(* IEC 61131-3 sources: ics/BLR101_ProenixContact/BLR101_5_ILC171_44/LogicalPOUs/MTR, 3 files *)

(* ---- MotorFB.ST ---- *)
(*@PROPERTIES_EX@
TYPE: POU
LOCALE: 0
IEC_LANGUAGE: ST
PLC_TYPE: independent
PROC_TYPE: independent
GROUP: MTRS.FB
*)
(*@KEY@:DESCRIPTION*)

(*@KEY@:END_DESCRIPTION*)
FUNCTION_BLOCK MotorFB

(*Group:Default*)

VAR_IN_OUT
	Mot_strct :	MTR;
	Aux_strct :	MTR_MISC;
END_VAR

VAR_INPUT
	Cycle :	CCL;
END_VAR

VAR_EXTERNAL
	TICK_1S_PLS :	BOOL;
END_VAR

VAR_OUTPUT
	Event :	MTR_EVENT;
END_VAR

(*@KEY@: WORKSHEET
NAME: MotorFB
IEC_LANGUAGE: ST
*)

if TICK_1S_PLS and not Aux_strct.AuxFlag then
	Aux_strct.Tick_1S:= true;
end_if;
Aux_strct.AuxFlag:= TICK_1S_PLS;

(*========================================================================================*)
	(*Alarm Feedback processing*)
(*========================================================================================*)
if Mot_strct.CW.Enable and ((Aux_strct.COM and not Mot_strct.SW.RUN) or (not Aux_strct.COM and Mot_strct.SW.RUN)) then
	if Aux_strct.Tick_1S then
		Aux_strct.AlrmTickCount:= Aux_strct.AlrmTickCount + 1;
	end_if;
else
	Aux_strct.AlrmTickCount:= 0;
end_if;

if Aux_strct.AlrmTickCount >= Aux_strct.SetOvertime then
	Aux_strct.AlarmFeedback:=true;
	Aux_strct.AlrmTickCount:= 0;
end_if;

if not Mot_strct.CW.ExtraEn and Aux_strct.COM then
	Aux_strct.AlarmBlock:= true;
end_if;

Mot_strct.SW.AlarmAccum:= Aux_strct.AlarmFeedback or Mot_strct.CW.ExtraAlarm or Aux_strct.AlarmBlock;

if Mot_strct.CW.ACK then
	Aux_strct.AlarmFeedback:=false;
	Aux_strct.AlarmBlock:= false;
end_if;

(*========================================================================================*)
	(*Auto/Manual mode selection*)
(*========================================================================================*)
if Mot_strct.CW.AutoMode then
	Mot_strct.SW.ManAuto:= true;
elsif Mot_strct.CW.ManMode then
	Mot_strct.SW.ManAuto:= false;
end_if;

Mot_strct.SW.ManOK:= not Mot_strct.SW.AlarmAccum and Mot_strct.CW.AuxON and Mot_strct.CW.Enable and not Mot_strct.SW.ManAuto;
Mot_strct.SW.AutoOK:= not Mot_strct.SW.AlarmAccum and Mot_strct.CW.AuxON and Mot_strct.CW.Enable and Mot_strct.SW.ManAuto;

(*========================================================================================*)
	(*Manual mode activation*)
(*========================================================================================*)

if Mot_strct.CW.ManStop or not Mot_strct.SW.ManOK then
	Mot_strct.SW.RunManual:=false;
elsif Mot_strct.CW.ManStart then
	Mot_strct.SW.RunManual:=true;
end_if;

(*========================================================================================*)
	(*Auto mode activation*)
(*========================================================================================*)
Mot_strct.SW.RunAuto:= Mot_strct.SW.AutoOK and Cycle.SW.Running;

(*========================================================================================*)
	(*Set command for start*)
(*========================================================================================*)
Aux_strct.COM:=((Mot_strct.SW.RunManual and Mot_strct.SW.ManOK) or (Mot_strct.SW.RunAuto and Mot_strct.SW.AutoOK and Mot_strct.CW.AutoON));
Mot_strct.SW.COM:=Aux_strct.COM and not Mot_strct.CW.SimEn;

(*========================================================================================*)
	(*Frequency limatation*)
(*========================================================================================*)
Mot_strct.MaxFreq:= LIMIT(0.0, Mot_strct.MaxFreq, 50.0);
Mot_strct.MinFreq:= LIMIT(0.0, Mot_strct.MinFreq, Mot_strct.MaxFreq);
Mot_strct.ManFreq:= LIMIT(Mot_strct.MinFreq, Mot_strct.ManFreq, Mot_strct.MaxFreq);
Mot_strct.AutoFreq:= LIMIT(Mot_strct.MinFreq, Mot_strct.AutoFreq, Mot_strct.MaxFreq);

if Mot_strct.SW.RunAuto and not Mot_strct.SW.AlarmAccum and Mot_strct.CW.AuxON then
	Aux_strct.SetValue:=Mot_strct.AutoFreq;
elsif not Mot_strct.SW.AlarmAccum and Mot_strct.SW.RunManual then
	Aux_strct.SetValue:=Mot_strct.ManFreq;
else
	Aux_strct.SetValue:=0.0;
end_if;

(*========================================================================================*)
	(*Work time counter*)
(*========================================================================================*)
if Mot_strct.SW.COM and Aux_strct.Tick_1S then
	Aux_strct.Seconds:= Aux_strct.Seconds + udint#1;
end_if;

Aux_strct.Minutes:= Aux_strct.Seconds / udint#60;
Aux_strct.Hours:= Aux_strct.Seconds / udint#3600;
Aux_strct.Days:= Aux_strct.Seconds / udint#86400;

(*========================================================================================*)
	(*Aux time counters*)
(*========================================================================================*)
if Aux_strct.CT1_ON and Aux_strct.Tick_1S then
	Aux_strct.CT1:= Aux_strct.CT1 + 1;
elsif not Aux_strct.CT1_ON then
	Aux_strct.CT1:= 0;
end_if;

if Aux_strct.CT2_ON and Aux_strct.Tick_1S then
	Aux_strct.CT2:= Aux_strct.CT2 + 1;
elsif not Aux_strct.CT2_ON then
	Aux_strct.CT2:= 0;
end_if;

(*========================================================================================*)
	(*Status processing*)
(*========================================================================================*)
if Mot_strct.SW.AlarmAccum then											(*Alarm*)
	Mot_strct.Status:=word#2;
elsif not Mot_strct.CW.ExtraEn then										(*Blocking*)
	Mot_strct.Status:=word#4;
elsif Mot_strct.SW.COM then												(*Working*)
	Mot_strct.Status:=word#1;
else																	(*Stoped*)
	Mot_strct.Status:=word#0;
end_if;

Mot_strct.CW.AutoMode:=false;
Mot_strct.CW.ManMode:=false;
Mot_strct.CW.ManStart:=false;
Mot_strct.CW.ManStop:=false;
Mot_strct.CW.ACK:=false;
Aux_strct.Tick_1S:= false;

(*================================================================================================*)
(*Motor Pulse Events*)
(*================================================================================================*)

Event.AlarmAccum:= false;
if Mot_strct.SW.AlarmAccum and not Aux_strct.EVENT_1 then
	Event.AlarmAccum:= true;
	Aux_strct.EVENT_1:= true;
elsif not Mot_strct.SW.AlarmAccum then
	Aux_strct.EVENT_1:= false;
end_if;
(*@KEY@: END_WORKSHEET *)
END_FUNCTION_BLOCK

(* ---- MTR.ST ---- *)
(*@PROPERTIES_EX@
TYPE: POU
LOCALE: 0
IEC_LANGUAGE: ST
PLC_TYPE: independent
PROC_TYPE: independent
GROUP: MTRS
*)
(*@KEY@:DESCRIPTION*)

(*@KEY@:END_DESCRIPTION*)
PROGRAM MTR

(*Group:Default*)

VAR_EXTERNAL
    M :	MOTOR;
    CCL :	CYCLE;
    WarnWord :	WRN;
    M_AUX :	MOTOR_MISC;
    AI :	SENSOR;
END_VAR

VAR
    i :	INT;
    j :	INT;
    PumpsFB :	MotorFB;
END_VAR

VAR_EXTERNAL
    MBRTU_Data :	MBRTU_SlvData;
END_VAR

VAR
    REAL_TO_MB :	REAL_TO_MB;
    y :	INT;
END_VAR

VAR_EXTERNAL
    MBTCP_Data :	MB_TCP_ARR_W_0_7167;
END_VAR

VAR
    y2 :	INT;
    y3 :	INT;
    y4 :	INT;
    y5 :	INT;
    y6 :	INT;
    y7 :	INT;
END_VAR

VAR_EXTERNAL
    M_EVENT :	MOTOR_EVENT;
END_VAR

(*@KEY@: WORKSHEET
NAME: MTR
IEC_LANGUAGE: ST
*)

    M[0].CW.AuxON			:= CCL[0].CW.AuxON and WarnWord.InputVoltage_1;
    M[1].CW.AuxON			:= CCL[0].CW.AuxON and WarnWord.InputVoltage_1;
    M[2].CW.AuxON			:= CCL[0].CW.AuxON and WarnWord.InputVoltage_1;
    M[3].CW.AuxON			:= CCL[0].CW.AuxON and WarnWord.InputVoltage_2;
    M[4].CW.AuxON			:= CCL[0].CW.AuxON and WarnWord.InputVoltage_2;

    M[0].ActFreq			:= AI[16].RealValue;
    M[1].ActFreq			:= AI[17].RealValue;
    M[2].ActFreq			:= AI[18].RealValue;
    M[3].ActFreq			:= AI[20].RealValue;
    M[4].ActFreq			:= AI[21].RealValue;

for i:= 0 to 4 do
(*================================================================================================*)
    (*Pumps 2.x structure parameters*)
(*================================================================================================*)
    M[i].CW.Enable			:= M[i].SW.Rem;
    M[i].CW.ExtraAlarm		:= M_AUX[i].DryMoveFault or M_AUX[i].DiffPressFault or M_AUX[i].TempFault;
    M[i].CW.ExtraEn			:= true;
    M[i].SW.RUN				:= M_AUX[i].DirRun or M_AUX[i].FCRun;
    M_AUX[i].SetOvertime	:= 30;

(*================================================================================================*)
    (*Pumps FB processing*)
(*================================================================================================*)
    PumpsFB(Mot_strct:=M[i],Aux_strct:=M_AUX[i],Cycle:=CCL[0]);
    M[i]:=PumpsFB.Mot_strct;
    M_AUX[i]:=PumpsFB.Aux_strct;
    M_EVENT[i]:=PumpsFB.Event;

(*================================================================================================*)
    (*Pumps 2.x FC parameters*)
(*================================================================================================*)
    j:= i + 13;
    M[i].Power				:= word_to_real(MBRTU_Data[i][0]) / 1000.0;
    M[i].Current			:= word_to_real(MBRTU_Data[i][2])/ 100.0;
    M[i].HeatSinkTemp		:= word_to_real(MBRTU_Data[i][4]);
    M[i].FC_StatusWord		:= MBRTU_Data[i][6];
    M[i].FC_AlarmWord		:= DW_TO_DWORD(MBRTU_Data[i][8],MBRTU_Data[i][9]);
    M[i].FC_WarnWord		:= DW_TO_DWORD(MBRTU_Data[i][10],MBRTU_Data[i][11]);

    M[i].RunHours           := dword_to_real(DW_TO_DWORD(MBRTU_Data[i][12],MBRTU_Data[i][13]));
    M[i].kWhCount			:= dword_to_real(DW_TO_DWORD(MBRTU_Data[i][14],MBRTU_Data[i][15]));

(*================================================================================================*)
    (*Reset and rewrite parameters to MB TCP*)
(*================================================================================================*)
    y:= i * 32 + 1700;
    y2:= y + 2;
    y3:= y + 3;
    y4:= y + 4;
    y5:= y + 5;
    y6:= y + 6;
    y7:= y + 7;

    REAL_TO_MB(IN:=M[i].MinFreq);
    MBTCP_Data[y2]:=REAL_TO_MB.LoWord;
    MBTCP_Data[y3]:=REAL_TO_MB.HiWord;

    REAL_TO_MB(IN:=M[i].MaxFreq);
    MBTCP_Data[y4]:=REAL_TO_MB.LoWord;
    MBTCP_Data[y5]:=REAL_TO_MB.HiWord;

    REAL_TO_MB(IN:=M[i].ManFreq);
    MBTCP_Data[y6]:=REAL_TO_MB.LoWord;
    MBTCP_Data[y7]:=REAL_TO_MB.HiWord;
end_for;

(*@KEY@: END_WORKSHEET *)
END_PROGRAM

(* ---- MTR_CTRL.ST ---- *)
(*@PROPERTIES_EX@
TYPE: POU
LOCALE: 0
IEC_LANGUAGE: ST
PLC_TYPE: independent
PROC_TYPE: independent
GROUP: MTRS
*)
(*@KEY@:DESCRIPTION*)

(*@KEY@:END_DESCRIPTION*)
PROGRAM MTR_CTRL

(*Group:Default*)

VAR
	RunPmpNum :	INT;
	TmpWTMax :	UDINT;
	TmpWTMin :	UDINT;
	TmpIndMax :	INT;
	TmpIndMin :	INT;
	i :	INT;
	StartPmpReq :	BOOL;
	StopPmpReq :	BOOL;
	Stage :	INT;
END_VAR

VAR_EXTERNAL
	CCL :	CYCLE;
END_VAR

VAR
	StartReqTmr :	TON;
	StopReqTmr :	TON;
	OverClckTmr :	TON;
	ReleaseTmr :	TON;
	TmpFreq :	REAL;
END_VAR

VAR_EXTERNAL
	M :	MOTOR;
	RGLTR :	REGULATOR;
	M_AUX :	MOTOR_MISC;
	MBTCP_Data :	MB_TCP_ARR_W_0_7167;
	AI :	SENSOR;
END_VAR

VAR
	MainPID :	FPID;
	TmpRotation :	BOOL;
	j :	INT;
END_VAR

VAR_EXTERNAL
	M_EVENT :	MOTOR_EVENT;
END_VAR

VAR
	TmpPmpAlarm :	BOOL;
	SysNum :	INT;
	LoInd :	INT;
	HiInd :	INT;
END_VAR

(*@KEY@: WORKSHEET
NAME: MTR_CTRL
IEC_LANGUAGE: ST
*)
(*================================================================================================*)
(*Work time sorting*)(*Number of working pumps evaluation*)(*PID min and max limits determination*)
(*================================================================================================*)
SysNum:= 0;																		(*Sequence number of cycle in cycles array (regulator in reg. array)*)
LoInd:= 0;																		(*First number of pump in pumps array used here*)
HiInd:= 4;																		(*Last number of pump in pumps array used here*)
RunPmpNum:= 0;
RGLTR[SysNum].LL:= 50.0;
RGLTR[SysNum].LH:= 0.0;

(*================================================================================================*)
for i:= LoInd to HiInd do

	if M[i].SW.AutoOK and M[i].SW.RUN then										(*Working pump number determination*)
		RunPmpNum:= RunPmpNum + 1;

		if M[i].MaxFreq > RGLTR[SysNum].LH  then								(*Assign pumps max. freq to RGLTR. hight limit*)
			RGLTR[SysNum].LH:= M[i].MaxFreq;
		end_if;

		if M[i].MinFreq < RGLTR[SysNum].LL then									(*Assign pumps min. freq to RGLTR. low limit*)
			RGLTR[SysNum].LL:= M[i].MinFreq;
		end_if;
	end_if;

	if not M[i].SW.AutoOK then
		M[i].CW.AutoON:= false;
	end_if;

	M[i].AutoFreq:= RGLTR[SysNum].Y / 10.0;										(*Assign pumps min. freq to RGLTR. low limit*)

(*================================================================================================*)
	(*Pumps Dry motion*)
(*================================================================================================*)
	j:= i * 2 + 2;

	M_AUX[i].CT1_ON:= (AI[j].RealValue <= 0.5) and M[i].SW.RUN and not M_AUX[i].DryMoveFault;

	if M_AUX[i].CT1 > 5 then
		M_AUX[i].DryMoveFault:= true;
	end_if;

	M_AUX[i].CT2_ON:= (AI[j].RealValue >= 1.0) and M_AUX[i].DryMoveFault;

	if M_AUX[i].CT2 > 30 then
		M_AUX[i].DryMoveFault:= false;
	end_if;

(*================================================================================================*)
	(*Alarm action*)
(*================================================================================================*)
	if M[i].SW.ManAuto and M_EVENT[i].AlarmAccum then
		TmpPmpAlarm:= true;
	end_if;
end_for;
(*================================================================================================*)

(*================================================================================================*)
	(*Set rotation command*)
(*================================================================================================*)
if CCL[SysNum].CW.Rotation then
	CCL[SysNum].SW.RotationON:= true;
	CCL[SysNum].CW.Rotation:= false;
end_if;

(*================================================================================================*)
	(*Start/Stop conditions*)
(*================================================================================================*)
StartReqTmr(IN:=(((RGLTR[SysNum].Y / 10.0) >= (RGLTR[SysNum].LH - 2.0)) and
				(RGLTR[SysNum].ActVal < RGLTR[SysNum].SP) and
				not StartPmpReq and CCL[SysNum].SW.Running),PT:=t#60s); 		(*Start auxiliary pump condition*)

StopReqTmr(IN:=(((RGLTR[SysNum].Y / 10.0) <= (RGLTR[SysNum].LL + 1.0)) and
				(RGLTR[SysNum].ActVal >= RGLTR[SysNum].SP) and
				not StopPmpReq and CCL[SysNum].SW.Running),PT:=t#60s);			(*Stop pump condition*)

(*================================================================================================*)
	(*Cycle handling*)
(*================================================================================================*)
IF CCL[SysNum].SW.Running then
	if (StartReqTmr.Q or (RunPmpNum < 1) or TmpPmpAlarm) and (Stage = 0) then	(*Stage route: 1 >> 2 >> 0*)
		Stage:= 1;
		if TmpPmpAlarm then
			TmpPmpAlarm:= false;
		end_if;
	elsif CCL[SysNum].SW.RotationON and (RunPmpNum > 0) and (Stage = 0) then	(*Stage route: 3 >> 1 >> 2 >> 4 >> 0*)
		TmpRotation:= true;
		Stage:= 3;
	elsif StopReqTmr.Q and (Stage = 0) then										(*Stage route: 3 >> 4 >> 0*)
		Stage:= 3;
	end_if;
else
	StartPmpReq:= false;
	StopPmpReq:= false;
	TmpFreq:= 0.0;
	CCL[SysNum].SW.RotationON:= false;
	TmpRotation:= false;
	Stage:= 0;
	TmpPmpAlarm:= false;

	for i:= LoInd to HiInd do
		M[i].CW.AutoON:= false;
	end_for;
end_if;

OverClckTmr(IN:=StartPmpReq and not OverClckTmr.Q,PT:=t#3s);					(*Overclocking pulse timer*)
ReleaseTmr(IN:=StopPmpReq and not ReleaseTmr.Q,PT:=t#3s);						(*Releasing pulse timer*)

case Stage of

	0:	StartPmpReq:= false;
		StopPmpReq:= false;
		TmpPmpAlarm:= false;
		CCL[SysNum].SW.RotationON:= false;
		TmpRotation:= false;
		TmpFreq:= 0.0;

	1:	StartPmpReq:= true;														(*Determ. higher work time*)
		TmpWTMin:= udint#0;
		TmpIndMin:= 0;
		for i:= LoInd to HiInd do
			if M_AUX[i].Seconds >= TmpWTMin then
				TmpWTMin:= M_AUX[i].Seconds;									(*Assign. higher work time to temporary var.*)
			end_if;
		end_for;

		for i:= LoInd to HiInd do
			if M[i].SW.AutoOK and not M[i].SW.RUN then							(*Determ. lowest work time pump*)
				if M_AUX[i].Seconds <= TmpWTMin then
					TmpWTMin:= M_AUX[i].Seconds;
					TmpIndMin:= i;												(*Determ. lowest work time pump index*)
				end_if;
			end_if;
		end_for;
		if (TmpIndMin < LoInd) and (TmpIndMin > HiInd) then
			Stage:= 5;
		else
			M[TmpIndMin].CW.AutoON:= true;										(*Start lowest work time pump*)
			TmpFreq:= M[TmpIndMin].MinFreq;										(*with min. frequency*)
			Stage:= 2;
		end_if;

	2:	M[TmpIndMin].AutoFreq:= TmpFreq;										(*Overclocking new pump*)
		if OverClckTmr.Q then
			TmpFreq:= TmpFreq + 1.0;
		elsif M[TmpIndMin].AutoFreq >= (RGLTR[SysNum].Y / 10.0)  then
			StartPmpReq:= false;
			if TmpRotation then
				Stage:= 4;
			else
				Stage:= 5;
			end_if;
		end_if;

	3:	TmpWTMax:= udint#0;														(*Determ. highest work time pump*)
		TmpIndMax:= 0;
		for i:= LoInd to HiInd do
			if M[i].SW.AutoOK and M[i].SW.RUN then
				if M_AUX[i].Seconds >= TmpWTMax then
					TmpWTMax:= M_AUX[i].Seconds;
					TmpIndMax:= i;
				end_if;
			end_if;
		end_for;
		if TmpRotation then
			Stage:= 1;
		else
			TmpFreq:= RGLTR[SysNum].Y / 10.0;
			Stage:= 4;
		end_if;

	4:	StopPmpReq:= true;														(*Releasing highest work time pump*)
		M[TmpIndMax].AutoFreq:= TmpFreq;
		if ReleaseTmr.Q then
			TmpFreq:= TmpFreq - 1.0;
		elsif M[TmpIndMax].AutoFreq <= M[TmpIndMax].MinFreq then
			M[TmpIndMax].CW.AutoON:= false;
			StopPmpReq:= false;
			Stage:= 5;
			TmpFreq:= 0.0;
		end_if;

	5:	StartPmpReq:= false;
		StopPmpReq:= false;
		TmpPmpAlarm:= false;
		CCL[SysNum].SW.RotationON:= false;
		TmpRotation:= false;
		TmpFreq:= 0.0;
		Stage:= 0;
end_case;

(*================================================================================================*)
	(*Main PID*)
(*================================================================================================*)
RGLTR[SysNum].ActVal:= AI[12].RealValue(* - AI[0].RealValue*);
MainPID(REMOTE:=CCL[SysNum].SW.Running,
		AUTO:=true,
		DIRECTN:=false,
		INTLCK:=(RunPmpNum <= 0),
		Tscan:=1.0,
		Yman:=RGLTR[SysNum].ManVal,
		SPR:=(RGLTR[SysNum].SP * 100.0),
		SPL:=0.0,
		X:=(RGLTR[SysNum].ActVal * 100.0),
		KP:=RGLTR[SysNum].Kp,
		TI:=RGLTR[SysNum].Tn,
		TD:=RGLTR[SysNum].Tv,
		HIGH:=(RGLTR[SysNum].LH * 10.0),
		LOW:=(RGLTR[SysNum].LL * 10.0),
		INTLCKV:=0.0);
RGLTR[SysNum].Y:=MainPID.Yout;

(*================================================================================================*)

(*@KEY@: END_WORKSHEET *)
END_PROGRAM
